// SIMATIC STEP 7 (V5.x) project TEMA 13 EJERCICIO 36
// CPU: CPU313 C-2 DP(1)
// station: P_ADR_BUS
// station: Hardware
// station: Equipo SIMATIC 300
// program: Programa S7(1)

SYMBOL_TABLE
"FLANCOS"	DB 1	DB 1
"MANIOBRA"	DB 2	DB 2
"P MARCHA"	I 0.0	BOOL
"F.C. C-LLENO"	I 0.1	BOOL
"F.C. C-REPOSO"	I 0.2	BOOL
"F.C C-VACIADO"	I 0.3	BOOL
"F.C. CT3 IZQUIERDA"	I 0.4	BOOL
"F.C. CT3 DERECHA"	I 0.5	BOOL
"P PARO"	I 0.6	BOOL
"Cycle Execution"	OB 1	OB 1
"CT1 M1"	Q 0.0	BOOL
"TRITURADOR M2"	Q 0.1	BOOL
"CT2 M3"	Q 0.2	BOOL
"M4 VOLCADO"	Q 0.3	BOOL
"M4 REPOSO"	Q 0.4	BOOL
"M5 CT3 DERECHA"	Q 0.5	BOOL
"M5 CT3 IZQUIERDA"	Q 0.6	BOOL
END_SYMBOL_TABLE

DATA_BLOCK "FLANCOS"	// DB 1
VERSION : 0.1
  STRUCT
   MO : BOOL ;
   M1 : BOOL ;
   M2 : BOOL ;
   M3 : BOOL ;
   M4 : BOOL ;
   M5 : BOOL ;
   M6 : BOOL ;
   M7 : BOOL ;
   M10 : BOOL ;
   M11 : BOOL ;
   M12 : BOOL ;
   M13 : BOOL ;
   M14 : BOOL ;
   M15 : BOOL ;
   M16 : BOOL ;
   M17 : BOOL ;
   M20 : BOOL ;
   M21 : BOOL ;
   M22 : BOOL ;
   M23 : BOOL ;
   M24 : BOOL ;
   M25 : BOOL ;
   M26 : BOOL ;
   M27 : BOOL ;
  END_STRUCT ;	
BEGIN
END_DATA_BLOCK

DATA_BLOCK "MANIOBRA"	// DB 2
VERSION : 0.1
  STRUCT
   M0 : BOOL ;
   M1 : BOOL ;
   M2 : BOOL ;
   M3 : BOOL ;
   M4 : BOOL ;
   M5 : BOOL ;
   M6 : BOOL ;
   M7 : BOOL ;
   M10 : BOOL ;
   M11 : BOOL ;
   M12 : BOOL ;
   M13 : BOOL ;
   M14 : BOOL ;
   M15 : BOOL ;
   M16 : BOOL ;
   M17 : BOOL ;
  END_STRUCT ;	
BEGIN
END_DATA_BLOCK

ORGANIZATION_BLOCK "Cycle Execution"	// OB 1
TITLE = "Main Program Sweep (Cycle)"
//TRITURADO Y TRANSPORTADO DE MATERIA PRIMA
VERSION : 0.1
VAR_TEMP
  OB1_EV_CLASS : BYTE ;	//Bits 0-3 = 1 (Coming event), Bits 4-7 = 1 (Event class 1)
  OB1_SCAN_1 : BYTE ;	//1 (Cold restart scan 1 of OB 1), 3 (Scan 2-n of OB 1)
  OB1_PRIORITY : BYTE ;	//Priority of OB Execution
  OB1_OB_NUMBR : BYTE ;	//1 (Organization block 1, OB1)
  OB1_RESERVED_1 : BYTE ;	//Reserved for system
  OB1_RESERVED_2 : BYTE ;	//Reserved for system
  OB1_PREV_CYCLE : INT ;	//Cycle time of previous OB1 scan (milliseconds)
  OB1_MIN_CYCLE : INT ;	//Minimum cycle time of OB1 (milliseconds)
  OB1_MAX_CYCLE : INT ;	//Maximum cycle time of OB1 (milliseconds)
  OB1_DATE_TIME : DATE_AND_TIME ;	//Date and time OB1 started
END_VAR
BEGIN
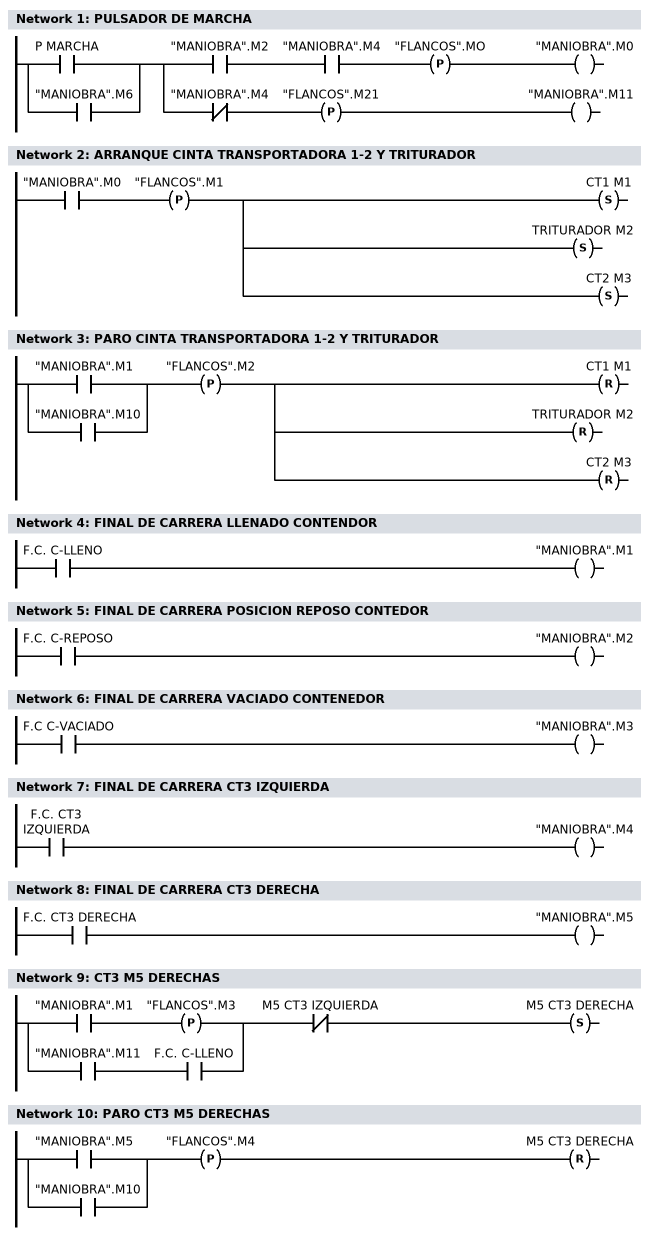
NETWORK
TITLE = PULSADOR DE MARCHA
      O     "P MARCHA";
      O     "MANIOBRA".M6;
      =     L 20.0;
      A     L 20.0;
      A     "MANIOBRA".M2;
      A     "MANIOBRA".M4;
      FP    "FLANCOS".MO;
      =     "MANIOBRA".M0;
      A     L 20.0;
      AN    "MANIOBRA".M4;
      FP    "FLANCOS".M21;
      =     "MANIOBRA".M11;
NETWORK
TITLE = ARRANQUE CINTA TRANSPORTADORA 1-2 Y TRITURADOR
      A     "MANIOBRA".M0;
      FP    "FLANCOS".M1;
      S     "CT1 M1";
      S     "TRITURADOR M2";
      S     "CT2 M3";
NETWORK
TITLE = PARO CINTA TRANSPORTADORA 1-2 Y TRITURADOR
      A(;
      O     "MANIOBRA".M1;
      O     "MANIOBRA".M10;
      );
      FP    "FLANCOS".M2;
      R     "CT1 M1";
      R     "TRITURADOR M2";
      R     "CT2 M3";
NETWORK
TITLE = FINAL DE CARRERA LLENADO CONTENDOR
//PARA CINTA 1-2 Y TRITURADOR Y ARRANCA CT3 DERECHAS
      A     "F.C. C-LLENO";
      =     "MANIOBRA".M1;
NETWORK
TITLE = FINAL DE CARRERA POSICION REPOSO CONTEDOR 
//EN REPOSO ESTARA PRESIONADO, ES DECIR CERRADO.PARA PODER PONER EN MARCHA EL 
//PROCESO EL CONTENEDOR TIENE QUE ESTAR EN REPOSO,YA QUE HAY QUE ASEGURARSE QUE 
//LA MATERIA PRIMA CAIGA EN EL CONTENEDOR. 
      A     "F.C. C-REPOSO";
      =     "MANIOBRA".M2;
NETWORK
TITLE = FINAL DE CARRERA VACIADO CONTENEDOR
//PARA LA RECOGIDA DEL CONTENEDOR 
      A     "F.C C-VACIADO";
      =     "MANIOBRA".M3;
NETWORK
TITLE = FINAL DE CARRERA CT3 IZQUIERDA
//EN REPOSO ESTARA PRESIONADO,COMPARTE ESTA FUNCION CON F.C REPOSO POR LA MISMA 
//RAZON Y ADEMAS PARA CT3 IZQUIERDA E INICIA EL PROCESO OTRA VEZ DE FORMA 
//INDEFINIDA. 
      A     "F.C. CT3 IZQUIERDA";
      =     "MANIOBRA".M4;
NETWORK
TITLE = FINAL DE CARRERA CT3 DERECHA
      A     "F.C. CT3 DERECHA";
      =     "MANIOBRA".M5;
NETWORK
TITLE = CT3 M5 DERECHAS
      A(;
      A     "MANIOBRA".M1;
      FP    "FLANCOS".M3;
      O;
      A     "MANIOBRA".M11;
      A     "F.C. C-LLENO";
      );
      AN    "M5 CT3 IZQUIERDA";
      S     "M5 CT3 DERECHA";
NETWORK
TITLE = PARO CT3 M5 DERECHAS
      A(;
      O     "MANIOBRA".M5;
      O     "MANIOBRA".M10;
      );
      FP    "FLANCOS".M4;
      R     "M5 CT3 DERECHA";
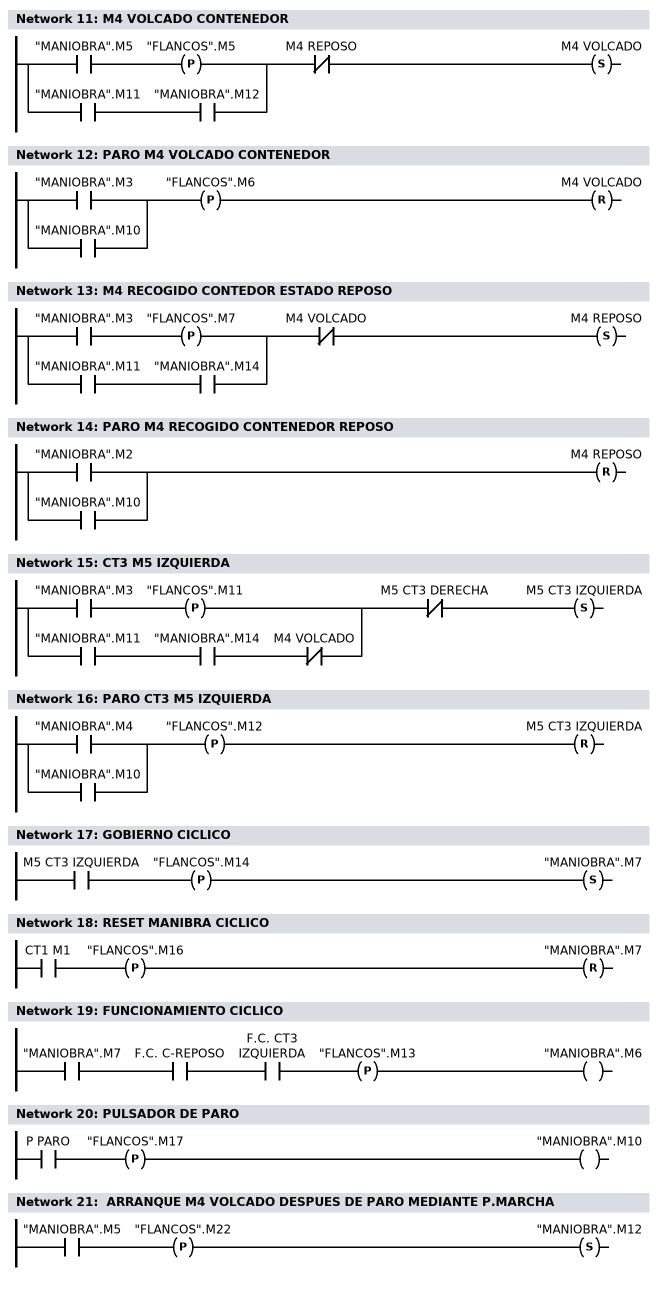
NETWORK
TITLE = M4 VOLCADO CONTENEDOR
      A(;
      A     "MANIOBRA".M5;
      FP    "FLANCOS".M5;
      O;
      A     "MANIOBRA".M11;
      A     "MANIOBRA".M12;
      );
      AN    "M4 REPOSO";
      S     "M4 VOLCADO";
NETWORK
TITLE = PARO M4 VOLCADO CONTENEDOR
      A(;
      O     "MANIOBRA".M3;
      O     "MANIOBRA".M10;
      );
      FP    "FLANCOS".M6;
      R     "M4 VOLCADO";
NETWORK
TITLE = M4 RECOGIDO CONTEDOR ESTADO REPOSO
      A(;
      A     "MANIOBRA".M3;
      FP    "FLANCOS".M7;
      O;
      A     "MANIOBRA".M11;
      A     "MANIOBRA".M14;
      );
      AN    "M4 VOLCADO";
      S     "M4 REPOSO";
NETWORK
TITLE = PARO M4 RECOGIDO CONTENEDOR REPOSO
      O     "MANIOBRA".M2;
      O     "MANIOBRA".M10;
      R     "M4 REPOSO";
NETWORK
TITLE = CT3 M5 IZQUIERDA
      A(;
      A     "MANIOBRA".M3;
      FP    "FLANCOS".M11;
      O;
      A     "MANIOBRA".M11;
      A     "MANIOBRA".M14;
      AN    "M4 VOLCADO";
      );
      AN    "M5 CT3 DERECHA";
      S     "M5 CT3 IZQUIERDA";
NETWORK
TITLE = PARO CT3 M5 IZQUIERDA
      A(;
      O     "MANIOBRA".M4;
      O     "MANIOBRA".M10;
      );
      FP    "FLANCOS".M12;
      R     "M5 CT3 IZQUIERDA";
NETWORK
TITLE = GOBIERNO CICLICO
//ESTA MARCA SERA LA ENCARGADA DE INDICAR LA POSICION A LA MAQUINA Y POR LO TANTO 
//INICIAR EL CICLO
      A     "M5 CT3 IZQUIERDA";
      FP    "FLANCOS".M14;
      S     "MANIOBRA".M7;
NETWORK
TITLE = RESET MANIBRA CICLICO
      A     "CT1 M1";
      FP    "FLANCOS".M16;
      R     "MANIOBRA".M7;
NETWORK
TITLE = FUNCIONAMIENTO CICLICO
//CUANDO TERMINE EL PROCESO VOLVERA A INICIAR LA SECUENCIA SIN NECESIDAD DE PULSAR
//EL P.MARCHA. 
      A     "MANIOBRA".M7;
      A     "F.C. C-REPOSO";
      A     "F.C. CT3 IZQUIERDA";
      FP    "FLANCOS".M13;
      =     "MANIOBRA".M6;
NETWORK
TITLE = PULSADOR DE PARO
//PARARA TODO EL PROCESO.EN EL CASO EXCEPCIONAL:
//ARRANQUE M5 CT3 DERECHAS-F.C.LLENADO CONTENEDOR ESTARA PRESIONADO Y NECISITA UN 
//PULSO DE P.MARCHA PARA SEGUIR EL PROCESO.
//ARRANQUE M4 VOLCADO CONTENEDOR-CONTACTO MARCA DE PARO P.MARCHA Y REANUDA.
//ARRANQUE M4 REPOSO CONTENEDOR-P.MARCHA ENVIARA EL IMPULSO NECESARIO PARA QUE 
//SIGA EL PROCES0 JUNTO CON EL CONTACTO CORRESPODIENTE DE PARO
//ARRANQUE M5 CT3 IZQUIERDAS-P. MARCHA  IGUAL QUE EL EL CASO ANTERIOR.
      A     "P PARO";
      FP    "FLANCOS".M17;
      =     "MANIOBRA".M10;
NETWORK
TITLE =  ARRANQUE M4 VOLCADO DESPUES DE PARO MEDIANTE P.MARCHA
      A     "MANIOBRA".M5;
      FP    "FLANCOS".M22;
      S     "MANIOBRA".M12;
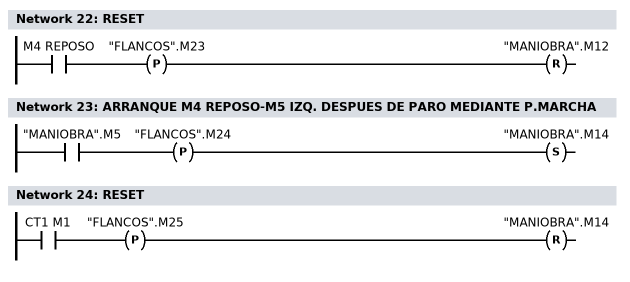
NETWORK
TITLE = RESET
      A     "M4 REPOSO";
      FP    "FLANCOS".M23;
      R     "MANIOBRA".M12;
NETWORK
TITLE = ARRANQUE M4 REPOSO-M5 IZQ. DESPUES DE PARO MEDIANTE P.MARCHA
      A     "MANIOBRA".M5;
      FP    "FLANCOS".M24;
      S     "MANIOBRA".M14;
NETWORK
TITLE = RESET
      A     "CT1 M1";
      FP    "FLANCOS".M25;
      R     "MANIOBRA".M14;
END_ORGANIZATION_BLOCK
